PROGRAM PRG_02_Xdrive
VAR
	TOF_horn: TOF;
	bRipCut: BOOL;
	signal_light_blink_fwd: FB_Blinker;
	signal_light_blink_rev: FB_Blinker;
	signal_light_blink1: FB_Blinker;
	signal_light_blink2: FB_Blinker;
	R_TRIG_2: R_TRIG;
	R_TRIG_3: R_TRIG;
	bRemoteDRV :BOOL;
	bRemoteREV :BOOL;
	TOF_0: TOF;
	TOF_1: TOF;
	F_TRIG_0: F_TRIG;
	F_TRIG_1: F_TRIG;
	TOF_XDriveBrakeDelay: TOF;


END_VAR
VAR // added by the converter: edge detectors and wires of the graphical bodies
    _w1, _w2 : BOOL;
END_VAR

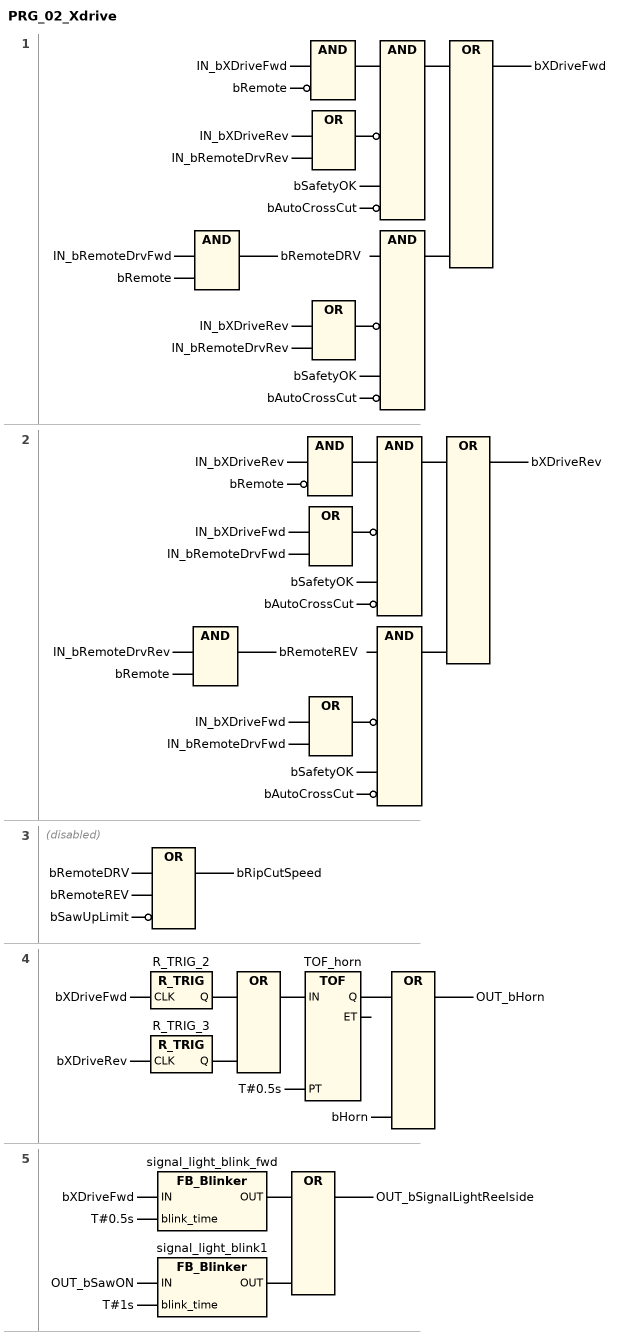
// NETWORK 1
_w1 := IN_bRemoteDrvFwd AND bRemote;
bRemoteDRV := _w1;
bXDriveFwd := (IN_bXDriveFwd AND NOT bRemote) AND NOT (IN_bXDriveRev OR IN_bRemoteDrvRev) AND bSafetyOK AND NOT bAutoCrossCut OR _w1 AND NOT (IN_bXDriveRev OR IN_bRemoteDrvRev) AND bSafetyOK AND NOT bAutoCrossCut;

// NETWORK 2
_w2 := IN_bRemoteDrvRev AND bRemote;
bRemoteREV := _w2;
bXDriveRev := (IN_bXDriveRev AND NOT bRemote) AND NOT (IN_bXDriveFwd OR IN_bRemoteDrvFwd) AND bSafetyOK AND NOT bAutoCrossCut OR _w2 AND NOT (IN_bXDriveFwd OR IN_bRemoteDrvFwd) AND bSafetyOK AND NOT bAutoCrossCut;

// NETWORK 3 (disabled)
// bRipCutSpeed := bRemoteDRV OR bRemoteREV OR NOT bSawUpLimit;

// NETWORK 4
R_TRIG_2(CLK := bXDriveFwd); // R_TRIG
R_TRIG_3(CLK := bXDriveRev); // R_TRIG
TOF_horn(IN := R_TRIG_2.Q OR R_TRIG_3.Q, PT := T#0.5s); // TOF
OUT_bHorn := TOF_horn.Q OR bHorn;

// NETWORK 5
signal_light_blink_fwd(IN := bXDriveFwd, blink_time := T#0.5s); // FB_Blinker
signal_light_blink1(IN := OUT_bSawON, blink_time := T#1s); // FB_Blinker
OUT_bSignalLightReelside := signal_light_blink_fwd.OUT OR signal_light_blink1.OUT;

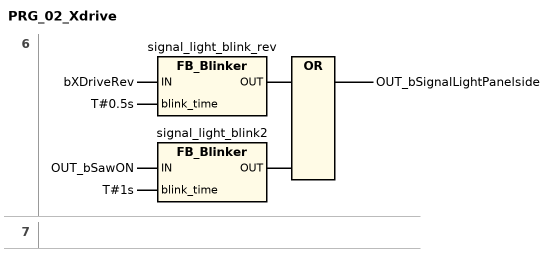
// NETWORK 6
signal_light_blink_rev(IN := bXDriveRev, blink_time := T#0.5s); // FB_Blinker
signal_light_blink2(IN := OUT_bSawON, blink_time := T#1s); // FB_Blinker
OUT_bSignalLightPanelside := signal_light_blink_rev.OUT OR signal_light_blink2.OUT;

// NETWORK 7

ACTION ACT_02_1_Xdrive:

// rRipCutSpeedSetting
END_ACTION

END_PROGRAM

(* stored: Version 1.1.0.1, ProductVersion 3.1.4024.15
   POU PRG_02_Xdrive: Id {a1053822-f050-4229-9728-e4ab6e39db5a}, SpecialFunc None
   Action ACT_02_1_Xdrive: Id {078b1921-ebc0-4435-bd35-7ea07ea778ac} *)
